FUNCTION_BLOCK fbDwordToReal
VAR_INPUT
	in_B0					: BYTE ;
	in_B1					: BYTE ;
	in_B2					: BYTE ;
	in_B3					: BYTE ;
	in_r_Res				: REAL ;
	in_i_Offset				: INT ;
END_VAR
VAR_OUTPUT
	out_r_Value				: REAL ;
END_VAR
VAR
	di_AddedValue			: DINT;
	r_Signed				: REAL;
	r_ResolutionResolved	: REAL;
END_VAR

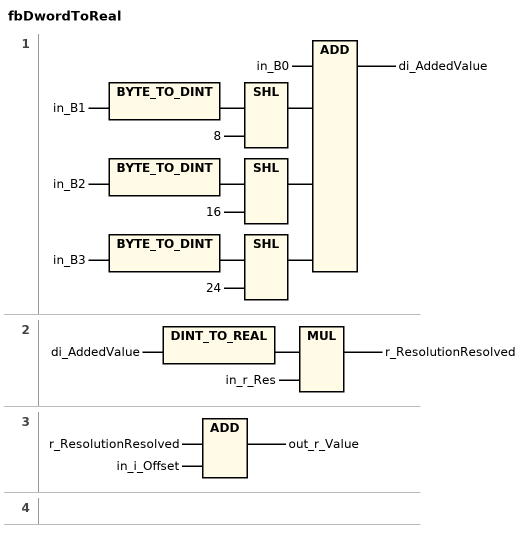
// NETWORK 1
di_AddedValue := in_B0 + SHL(BYTE_TO_DINT(in_B1), 8) + SHL(BYTE_TO_DINT(in_B2), 16) + SHL(BYTE_TO_DINT(in_B3), 24);

// NETWORK 2
r_ResolutionResolved := DINT_TO_REAL(di_AddedValue) * in_r_Res;

// NETWORK 3
out_r_Value := r_ResolutionResolved + in_i_Offset;

// NETWORK 4

END_FUNCTION_BLOCK

(* stored: Version 1.1.0.1, ProductVersion 3.1.4024.12
   POU fbDwordToReal: Id {a2627284-4b12-425a-8b5a-3beb64366992}, SpecialFunc None *)
